PROGRAM MAIN
VAR
	FB_Axis_X1 	: 	FB_Axis;
	st_Axis_X1	: 	ST_AxisStruct;
	
//	FB_Axis_X2 	: 	FB_Axis;
//	FB_Axis_Y 	: 	FB_Axis;
//	FB_Axis_Z 	: 	FB_Axis;
END_VAR

//st_Axis_X1.stControl.bEnable := TRUE;
st_Axis_X1.stStatus.bFwEnabled := TRUE;
st_Axis_X1.stStatus.bBwEnabled := TRUE;
FB_Axis_X1(stAxisStruct:= st_Axis_X1 );

END_PROGRAM

(* stored: Version 1.1.0.1, ProductVersion 3.1.4024.5
   POU MAIN: Id {ccac79b0-c6a0-4f9e-89fe-3f9f18cda55f}, SpecialFunc None *)
